FUNCTION_BLOCK FB_MicroStepCountTest
VAR_INPUT
	bExecute: BOOL;
	fStart: LREAL;
	fEnd: LREAL;
	fIncr: LREAL;
	fTheoryStep: LREAL;
END_VAR
VAR_OUTPUT
	bDone: BOOL;
	nPosCount: INT := -1;
	nTheoryCount: DINT;
	nSteps: INT := -1;
	nMissedSteps: INT;
	nMaxMissCombo: INT;
	fStepPercent: LREAL;
END_VAR
VAR_IN_OUT
	Axis: AXIS_REF;
END_VAR
VAR
	fbMoveStart: MC_MoveAbsolute;
	fbStep: MC_MoveRelative;
	fbSettleTimer: TON;
	bStarted: BOOL;
	bTimerLatch: BOOL;
	bDoStep: BOOL;
	nWaitCount: UINT;
	fLastPosition: LREAL;
	nMissCombo: INT;
	nOldTheoryCount: DINT;
END_VAR

// Goal: Move axis slightly, repeatedly, and see how many effective positions we have between two given positions.
// Works best if fIncr is greater than the encoder noise but less than the smallest theoretical step
fbMoveStart(Axis:=Axis,
	Execute:=bExecute AND NOT bStarted AND NOT bDone,
	Position:=fStart,
	Velocity:=1);
fbStep(Axis:=Axis,
	Execute:=bDoStep AND bStarted AND NOT bDone,
	Distance:=fIncr,
	Velocity:=1);
fbSettleTimer(IN:=fbMoveStart.Done OR fbStep.Done,
	PT:=T#2S);
IF fbSettleTimer.Q THEN
	IF NOT bStarted THEN
		bDoStep := TRUE;
	END_IF
	bStarted := TRUE;
	bTimerLatch := TRUE;
	nSteps := nSteps + 1;
	nOldTheoryCount := nTheoryCount;
	nTheoryCount := TRUNC((Axis.NcToPlc.ActPos - fStart)/fTheoryStep);
	IF Axis.NcToPlc.ActPos >= fLastPosition + fIncr THEN
		fLastPosition := Axis.NcToPlc.ActPos;
		nPosCount := nPosCount + 1;
		nMissCombo := 0;
	ELSIF nTheoryCount - nOldTheoryCount >= 1 THEN
		nMissedSteps := nMissedSteps + 1;
		nMissCombo := nMissCombo + 1;
		IF nMissCombo > nMaxMissCombo THEN
			nMaxMissCombo := nMissCombo;
		END_IF
	END_IF
	IF nTheoryCount > 0 THEN
		fStepPercent := 100 * nPosCount / nTheoryCount;
	END_IF
	IF fLastPosition >= fEnd THEN
		bDone := TRUE;
	END_IF
END_IF
IF bTimerLatch THEN
	bTimerLatch := bDoStep;
	bDoStep := NOT bDoStep;
END_IF

END_FUNCTION_BLOCK

(* stored: Version 1.1.0.1, ProductVersion 3.1.4020.14
   POU FB_MicroStepCountTest: Id {d12fc184-7092-47a4-94e5-3a29711f3d42}, SpecialFunc None *)
